TYPE CuBaseRecurringFail :
STRUCT
	Reached:BOOL;
	Result:TcoComprehensiveResult;
	Counter:UINT;
	
	
	
	
	
END_STRUCT
END_TYPE

(* stored: Version 1.1.0.1
   DUT CuBaseRecurringFail: Id {8ab05726-cba0-0d91-3c67-9c8300ca4e23} *)
